(* CoDeSys 2.3.9.37 project: AscensorCompleto.pro *)
(* Libraries: Standard.lib 4.10.05 12:14:46, IecSfc.lib 13.4.06 16:51:28 *)

(* Global variable list: Global_Variables *)
VAR_GLOBAL
   (*Entradas *)
      (* Sensores de posición en plantas *)
      S0: BOOL;
      S1: BOOL;
      S2: BOOL;
      S3: BOOL;
      (* Pulsadores de llamadas en planta *)
      P0: BOOL;
      P1: BOOL;
      P2: BOOL;
      P3: BOOL;
     (* Pulsadores en cabina *)
      C0: BOOL;
      C1: BOOL;
      C2: BOOL;
      C3: BOOL;
   (*Salidas *)
      Motor_arriba : BOOL;
      Motor_Abajo : BOOL;
    (* luces asociadas a los pulsadores. Se usarán
        si se quiere implementar memoria de llamada *)
     LuzP0:BOOL;
     LuzP1:BOOL;
     LuzP2:BOOL;
     LuzP3:BOOL;
    LuzC0:BOOL;
     LuzC1:BOOL;
     LuzC2:BOOL;
     LuzC3:BOOL;
END_VAR

(* POU PLC_PRG, ST *)
PROGRAM PLC_PRG
VAR
END_VAR
Movimiento;
END_PROGRAM

(* POU Movimiento, ST *)
PROGRAM Movimiento
VAR
    pos:INT:=0;
END_VAR
IF (Motor_arriba AND pos>=-240) THEN
   pos:=pos-2;
END_IF


IF (Motor_abajo AND pos<=-2) THEN
   pos:=pos+2;
END_IF

IF (pos>=0 AND pos<=2) THEN
  S0:=TRUE;
ELSE
  S0:=FALSE;
END_IF

IF (pos>=-78 AND pos<=-74) THEN
  S1:=TRUE;
ELSE
  S1:=FALSE;
END_IF

IF (pos>=-156 AND pos<=-152) THEN
  S2:=TRUE;
ELSE
  S2:=FALSE;
END_IF

IF (pos>=-242 AND pos<=-240) THEN
  S3:=TRUE;
ELSE
  S3:=FALSE;
END_IF
END_PROGRAM

(* Visualisation Ascensor
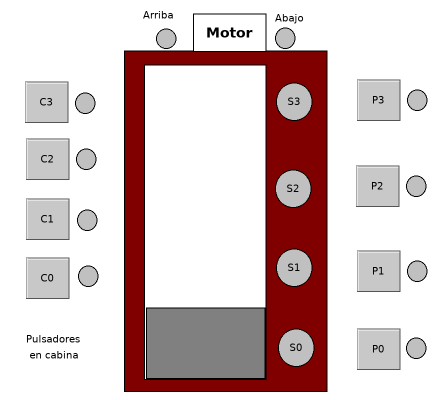
ellipse at (285,341)-(321,379): text "S0"; alarm colour if S0
ellipse at (283,261)-(319,299): text "S1"; alarm colour if S1
ellipse at (282,182)-(318,220): text "S2"; alarm colour if S2
ellipse at (283,95)-(319,133): text "S3"; alarm colour if S3
rounded rectangle at (153,320)-(272,391): y offset Movimiento.pos
button at (364,341)-(407,382): text "P0"; taps P0
button at (364,263)-(407,304): text "P1"; taps P1
button at (363,178)-(406,219): text "P2"; taps P2
button at (364,92)-(407,133): text "P3"; taps P3
rectangle at (200,26)-(273,64): text "Motor"
ellipse at (163,41)-(183,61): alarm colour if Motor_arriba
ellipse at (282,40)-(302,61): alarm colour if Motor_abajo
rectangle at (138,18)-(193,37): text "Arriba"
rectangle at (269,21)-(324,40): text "Abajo"
rectangle at (22,329)-(98,374): text "Pulsadores"
rectangle at (23,345)-(99,390): text "en cabina"
button at (33,270)-(76,311): text "C0"; taps C0
button at (33,211)-(76,252): text "C1"; taps C1
button at (33,151)-(76,192): text "C2"; taps C2
button at (32,94)-(75,135): text "C3"; taps C3
ellipse at (414,102)-(434,123): alarm colour if LuzP3
ellipse at (413,188)-(433,209): alarm colour if LuzP2
ellipse at (414,273)-(434,294): alarm colour if LuzP1
ellipse at (413,350)-(433,371): alarm colour if LuzP0
ellipse at (82,105)-(102,126): alarm colour if LuzC3
ellipse at (83,161)-(103,182): alarm colour if LuzC2
ellipse at (84,222)-(104,243): alarm colour if LuzC1
ellipse at (85,278)-(105,299): alarm colour if LuzC0
3 more shapes without text or variables
*)
